// TIA Portal V20 export
TYPE "LWONIK_typeScsMode"
// stored: Access Published
   STRUCT
      Disabled : Bool;
      PendantReq : Bool;
      setup : Bool;
      auto : Bool;
      disable : Bool;
   END_STRUCT;
END_TYPE
